// TIA Portal V17 export
// export: Created 2025-06-26T07:49:18.8669555Z, ExportSetting WithDefaults, DisplayName Totally Integrated Automation Portal, DisplayVersion V17 Update 8, DisplayName TIA Portal Openness, DisplayVersion V17 Update 8, DisplayName TIA Portal Version Control Interface, DisplayVersion V17, DisplayName STEP 7 Professional, DisplayVersion V17 Update 8, DisplayName STEP 7 Safety, DisplayVersion V17 Update 6, DisplayName WinCC Advanced, DisplayVersion V17 Update 8
TYPE "typeDataPtr"
// stored: IsFailsafeCompliant false
   STRUCT
      data : Array[0..7] of Word;
   END_STRUCT;
END_TYPE
